FUNCTION atan2 : LREAL
VAR_INPUT
	y,x:lreal;
END_VAR
VAR
END_VAR

IF(x>0)THEN
	atan2:=ATAN(y/x);
ELSIF(x<0 AND y>=0)THEN
	atan2:=ATAN(y/x)+PI;
ELSIF(x<0 AND y<0)THEN
	atan2:=ATAN(y/x)-PI;
ELSIF(x=0 AND y>0)THEN
	atan2:=PI/2;
ELSIF(x=0 AND y<0)THEN
	atan2:=-1*PI/2;
END_IF

END_FUNCTION

(* stored: Version 1.1.0.1, ProductVersion 3.1.4024.12
   POU atan2: Id {18a456ff-3b8c-4dc0-9e21-09d01c458edb}, SpecialFunc None *)
